// TIA Portal V20 export
FUNCTION "P100" : Void   // FC20, FBD
{ S7_Optimized_Access := 'TRUE' }
// stored: SetENOAutomatically false
   VAR_TEMP
      Temp : "DigVal";
      Temp_1 : "DigVal";
      Temp_3 : "DigVal";
      Temp_2 : "DigVal";
      Temp_Error : "DigVal";
      Intlock : "DigVal";
      Intlock_In : "DigVal";
      State : "Service_States";
   END_VAR
BEGIN

REGION Network 1: Channel input
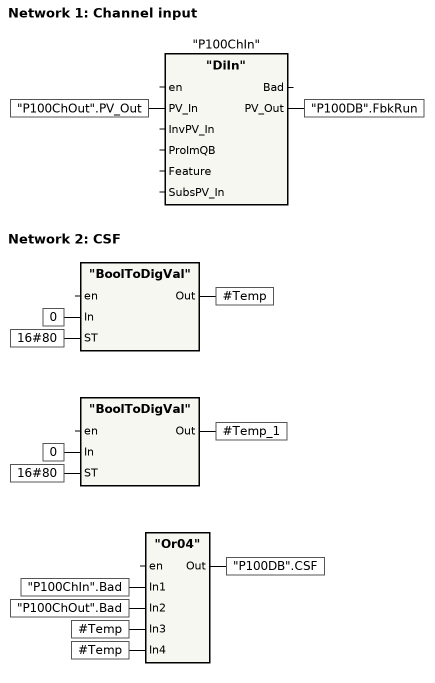
   "P100ChIn"(PV_In := "P100ChOut".PV_Out, PV_Out => "P100DB".FbkRun);   // "DiIn"
END_REGION

REGION Network 2: CSF
   "BoolToDigVal"(In := 0, ST := 16#80, Out => #Temp);
   "BoolToDigVal"(In := 0, ST := 16#80, Out => #Temp_1);
   "Or04"(In1 := "P100ChIn".Bad, In2 := "P100ChOut".Bad, In3 := #Temp, In4 := #Temp, Out => "P100DB".CSF);
END_REGION

REGION Network 3: Interlock
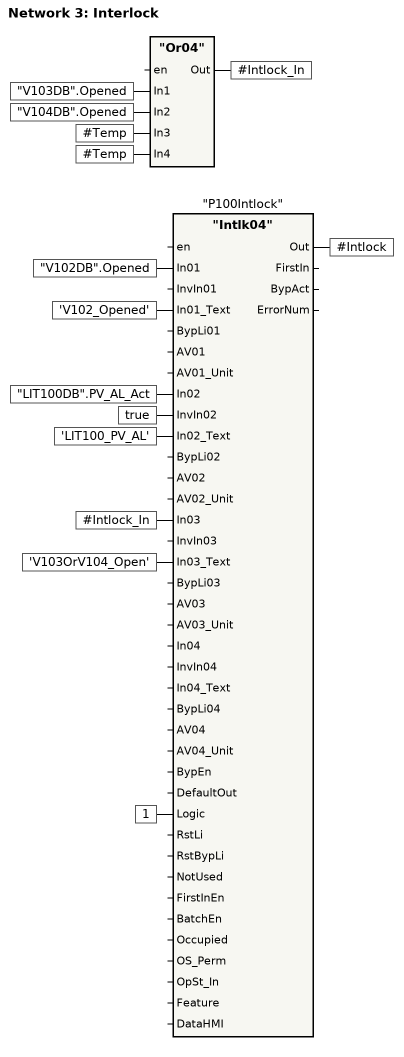
   "Or04"(In1 := "V103DB".Opened, In2 := "V104DB".Opened, In3 := #Temp, In4 := #Temp, Out => #Intlock_In);
   "P100Intlock"(In01 := "V102DB".Opened,   // "Intlk04"
                 In01_Text := 'V102_Opened',
                 In02 := "LIT100DB".PV_AL_Act,
                 InvIn02 := true,
                 In02_Text := 'LIT100_PV_AL',
                 In03 := #Intlock_In,
                 In03_Text := 'V103OrV104_Open',
                 Logic := 1,
                 Out => #Intlock);
END_REGION

REGION Network 4: MotL
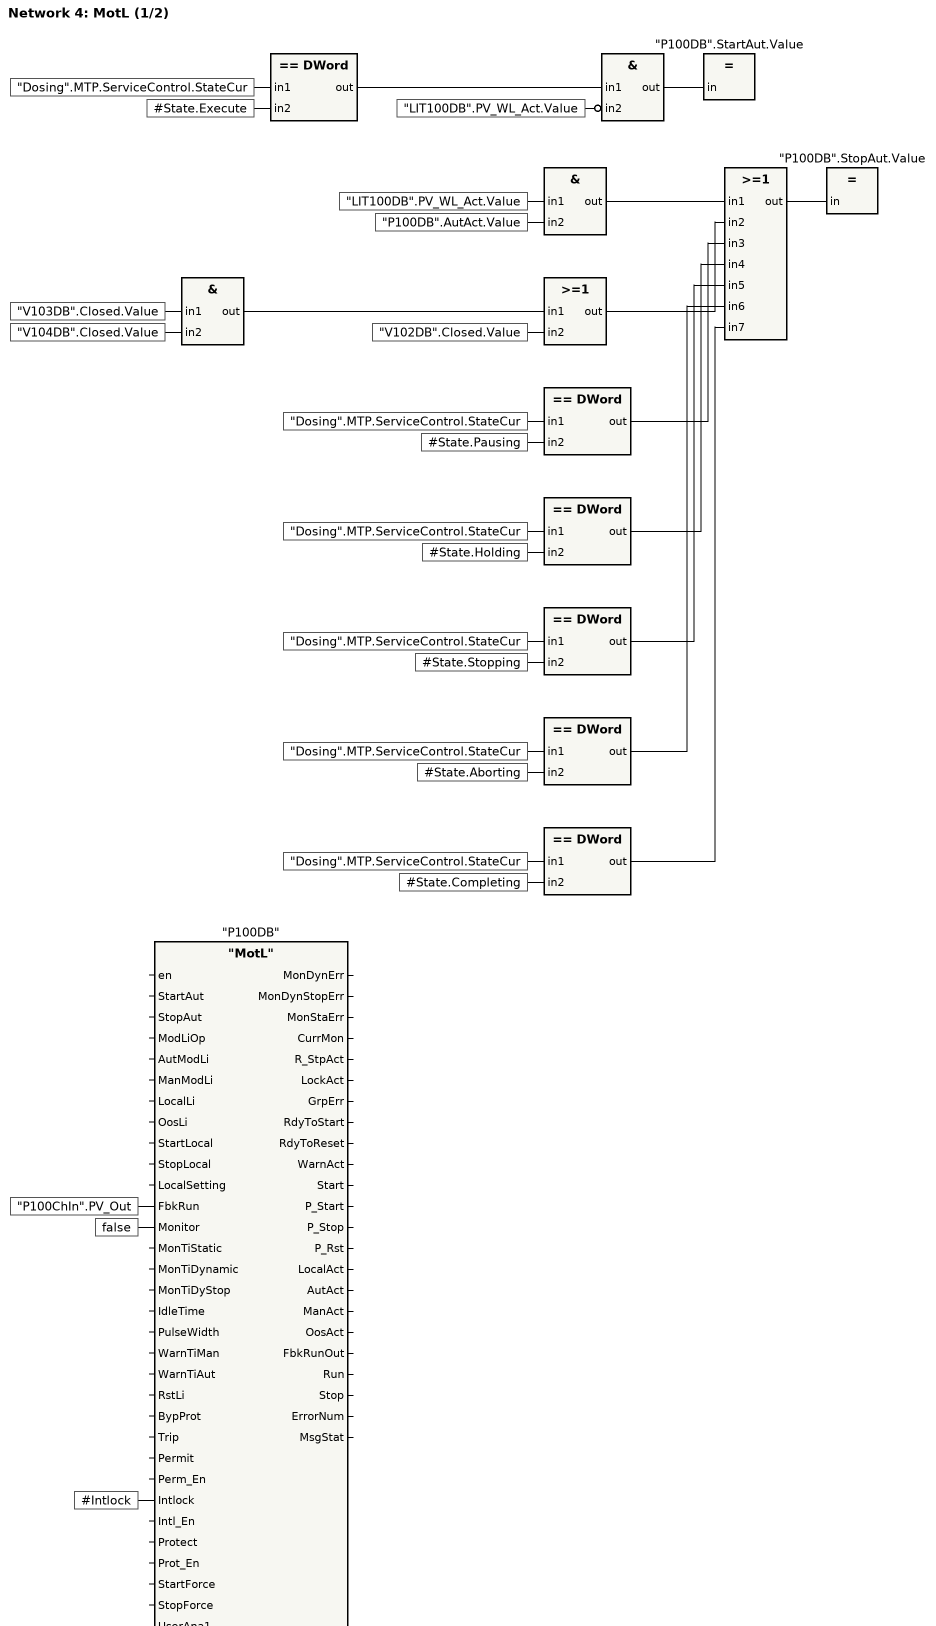
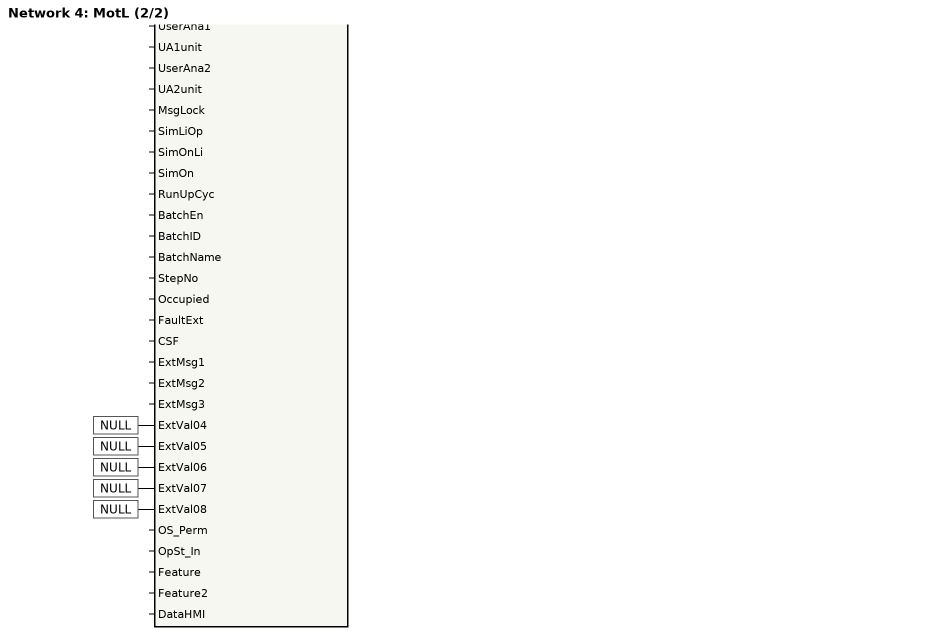
   "P100DB".StartAut.Value := ("Dosing".MTP.ServiceControl.StateCur = #State.Execute) AND NOT "LIT100DB".PV_WL_Act.Value;
   "P100DB".StopAut.Value := ("LIT100DB".PV_WL_Act.Value AND "P100DB".AutAct.Value) OR ("V103DB".Closed.Value AND "V104DB".Closed.Value) OR "V102DB".Closed.Value OR ("Dosing".MTP.ServiceControl.StateCur = #State.Pausing) OR ("Dosing".MTP.ServiceControl.StateCur = #State.Holding) OR ("Dosing".MTP.ServiceControl.StateCur = #State.Stopping) OR ("Dosing".MTP.ServiceControl.StateCur = #State.Aborting) OR ("Dosing".MTP.ServiceControl.StateCur = #State.Completing);
   "P100DB"(FbkRun := "P100ChIn".PV_Out,   // "MotL"
            Monitor := false,
            Intlock := #Intlock,
            ExtVal04 := NULL,
            ExtVal05 := NULL,
            ExtVal06 := NULL,
            ExtVal07 := NULL,
            ExtVal08 := NULL);
END_REGION

REGION Network 5: MTP
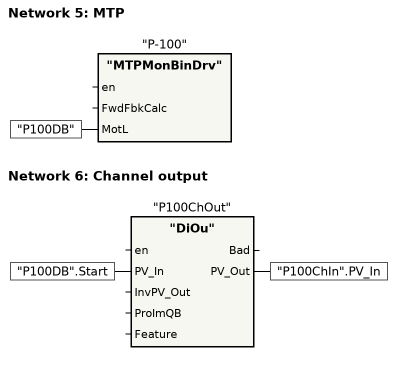
   "P-100"(MotL := "P100DB");   // "MTPMonBinDrv"
END_REGION

REGION Network 6: Channel output
   "P100ChOut"(PV_In := "P100DB".Start, PV_Out => "P100ChIn".PV_In);   // "DiOu"
END_REGION
END_FUNCTION
